// TIA Portal V17 program export: 1 tag tables, 0 data types, 4 data blocks, 2 code blocks (in call order from the OBs), 2 instance data blocks

VAR_GLOBAL   // PLC tag table "Tabla de variables estándar"
   System_Byte AT %MB1 : Byte;
   FirstScan AT %M1.0 : Bool;
   DiagStatusUpdate AT %M1.1 : Bool;
   AlwaysTRUE AT %M1.2 : Bool;
   AlwaysFALSE AT %M1.3 : Bool;
   Clock_Byte AT %MB0 : Byte;
   Clock_10Hz AT %M0.0 : Bool;
   Clock_5Hz AT %M0.1 : Bool;
   "Clock_2.5Hz" AT %M0.2 : Bool;
   Clock_2Hz AT %M0.3 : Bool;
   "Clock_1.25Hz" AT %M0.4 : Bool;
   Clock_1Hz AT %M0.5 : Bool;
   "Clock_0.625Hz" AT %M0.6 : Bool;
   "Clock_0.5Hz" AT %M0.7 : Bool;
   RISING_EDGE AT %M3.0 : Bool;
   INDEX AT %MB2 : USInt;
   MODE AT %MB6 : USInt;
   RISING_REQ AT %M3.1 : Bool;
   VOLTS AT %MW4 : UInt;
   AMPS AT %MW8 : UInt;
   HERTZ AT %MW10 : UInt;
   RPM AT %MW12 : UInt;
END_VAR
VAR_GLOBAL CONSTANT   // user constants
   READ : USInt := 0;
   WRITE : USInt := 1;
END_VAR

DATA_BLOCK "DB_MB_COMM_LOAD"   // DB4
{ S7_Optimized_Access := 'TRUE' }
VERSION : 0.1
// stored: AutoNumber true, DBAccessibleFromOPCUA true, IsOnlyStoredInLoadMemory false, IsRetainMemResEnabled false, IsWriteProtectedInAS false, MemoryReserve 100
   VAR
      COMM_DONE : Bool;
      COMM_ERROR : Bool;
      COMM_STATUS : Word;
   END_VAR
BEGIN
END_DATA_BLOCK

DATA_BLOCK "DB_ADDR"   // DB5
{ S7_Optimized_Access := 'FALSE' }
VERSION : 0.1
// stored: AutoNumber true, DBAccessibleFromOPCUA true, IsOnlyStoredInLoadMemory false, IsWriteProtectedInAS false
   VAR
      VOLT : UDInt := 48455;
      AMP : UDInt := 48453;
      FRE : UDInt := 48452;
      RPM : UDInt := 48456;
      SPEED : UDInt := 42331;
      RUN : UDInt := 42332;
      DIR : UDInt := 42333;
      OUT : UDInt;
   END_VAR
BEGIN
END_DATA_BLOCK

DATA_BLOCK "DB_GS1_MODBUS"   // DB6
{ S7_Optimized_Access := 'TRUE' }
VERSION : 0.1
// stored: AutoNumber true, DBAccessibleFromOPCUA true, IsOnlyStoredInLoadMemory false, IsRetainMemResEnabled false, IsWriteProtectedInAS false, MemoryReserve 100
   VAR
      GS1_DONE : Bool;
      GS1_BUSY : Bool;
      GS1_ERROR : Bool;
      GS1_STATUS : Word;
   END_VAR
BEGIN
END_DATA_BLOCK

DATA_BLOCK "DB_RW_PAR"   // DB3
{ S7_Optimized_Access := 'FALSE' }
VERSION : 0.1
// stored: AutoNumber true, DBAccessibleFromOPCUA true, IsOnlyStoredInLoadMemory false, IsWriteProtectedInAS false
   VAR
      VOLT_ACT : UInt;
      AMP_ACT : UInt;
      FRE_ACT : UInt;
      RPM_ACT : UInt;
      "SPEED(FREQ)" : UInt := 0;
      RUN : UInt := 0;
      DIR : UInt := 0;
      OUT : UInt;
   END_VAR
BEGIN
END_DATA_BLOCK

ORGANIZATION_BLOCK "Main"   // OB1, LAD, ProgramCycle
TITLE = "Main Program Sweep (Cycle)"
{ S7_Optimized_Access := 'TRUE' }
VERSION : 0.1
// stored: AutoNumber true, IsIECCheckEnabled false, SetENOAutomatically false
   VAR_INPUT
      Initial_Call : Bool;   // Initial call of this OB
      Remanence : Bool;   // =True, if remanent data are available
   END_VAR
BEGIN

REGION Network 1: ----------[MODBUS COMMUNICATION SETTING UP]----------
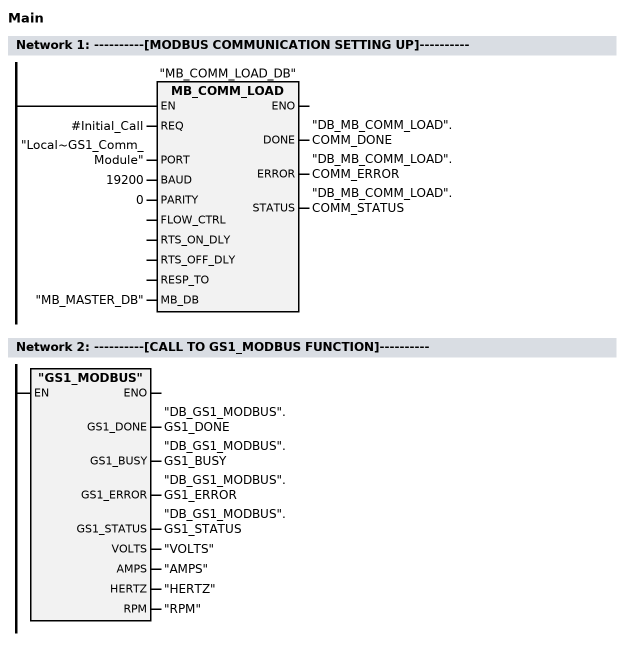
   RUNG wire#powerrail
      "MB_COMM_LOAD_DB".MB_COMM_LOAD(REQ := #Initial_Call, PORT := "Local~GS1_Comm_Module", BAUD := 19200, PARITY := 0, FLOW_CTRL :=, RTS_ON_DLY :=, RTS_OFF_DLY :=, RESP_TO :=, MB_DB := "MB_MASTER_DB", DONE => "DB_MB_COMM_LOAD".COMM_DONE, ERROR => "DB_MB_COMM_LOAD".COMM_ERROR, STATUS => "DB_MB_COMM_LOAD".COMM_STATUS)
   END_RUNG
   // the same network as SCL:
   "MB_COMM_LOAD_DB"(REQ := #Initial_Call,   // MB_COMM_LOAD
                     PORT := "Local~GS1_Comm_Module",
                     BAUD := 19200,
                     PARITY := 0,
                     MB_DB := "MB_MASTER_DB",
                     DONE => "DB_MB_COMM_LOAD".COMM_DONE,
                     ERROR => "DB_MB_COMM_LOAD".COMM_ERROR,
                     STATUS => "DB_MB_COMM_LOAD".COMM_STATUS);
END_REGION

REGION Network 2: ----------[CALL TO GS1_MODBUS FUNCTION]----------
   RUNG wire#powerrail
      "GS1_MODBUS"(GS1_DONE => "DB_GS1_MODBUS".GS1_DONE, GS1_BUSY => "DB_GS1_MODBUS".GS1_BUSY, GS1_ERROR => "DB_GS1_MODBUS".GS1_ERROR, GS1_STATUS => "DB_GS1_MODBUS".GS1_STATUS, VOLTS => "VOLTS", AMPS => "AMPS", HERTZ => "HERTZ", RPM => "RPM")
   END_RUNG
   // the same network as SCL:
   "GS1_MODBUS"(GS1_DONE => "DB_GS1_MODBUS".GS1_DONE,
                GS1_BUSY => "DB_GS1_MODBUS".GS1_BUSY,
                GS1_ERROR => "DB_GS1_MODBUS".GS1_ERROR,
                GS1_STATUS => "DB_GS1_MODBUS".GS1_STATUS,
                VOLTS => "VOLTS",
                AMPS => "AMPS",
                HERTZ => "HERTZ",
                RPM => "RPM");
END_REGION
END_ORGANIZATION_BLOCK

FUNCTION "GS1_MODBUS" : Void   // FC1, LAD
TITLE = FUNCTION FOR SEND THE MODE (R/W OF REGISTERS), MODBUS MODE, REGISTERS ADDRESS AND LOAD VALUES
{ S7_Optimized_Access := 'TRUE' }
VERSION : 0.1
// stored: AutoNumber true, IsIECCheckEnabled false, SetENOAutomatically false, UDAEnableTagReadback false
   VAR_OUTPUT
      GS1_DONE : Bool;
      GS1_BUSY : Bool;
      GS1_ERROR : Bool;
      GS1_STATUS : Word;
      VOLTS : UInt;
      AMPS : UInt;
      HERTZ : UInt;
      RPM : UInt;
   END_VAR
   VAR_TEMP
      RW : Int;
   END_VAR
   VAR_TEMP   // added for the SCL form of the ladder/FBD networks
      _w1 : Bool;
   END_VAR
BEGIN

REGION Network 1: ----------[GENERATE MODBUS ADDRESS & COMMAND DATA INDEX]----------
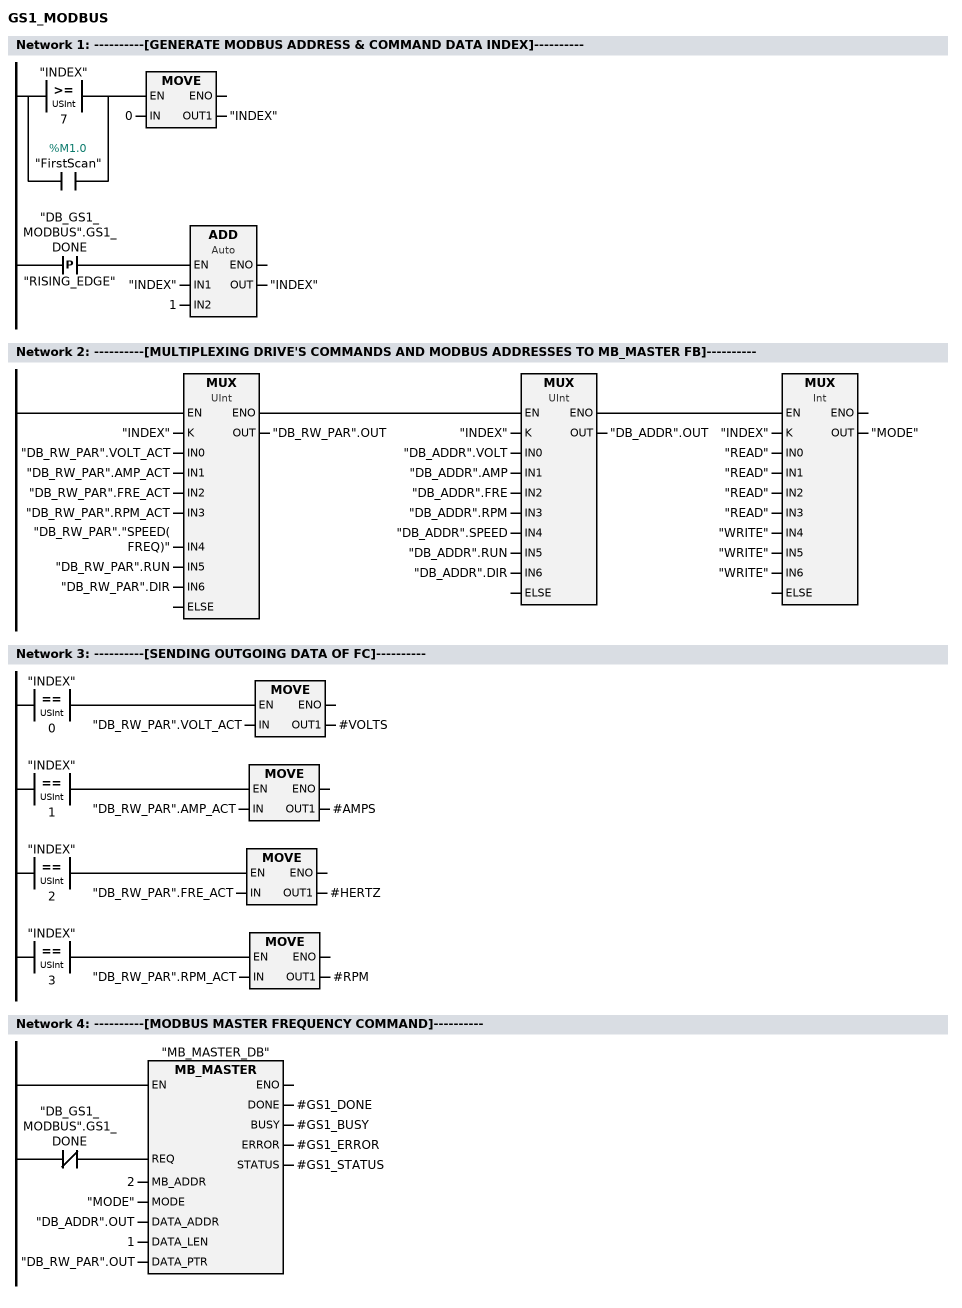
   RUNG wire#powerrail
      { S7_Templates := "SrcType := USInt" } GE_Contact(in1 := "INDEX", in2 := 7)
      wire#w1
      Move(in := 0, out1 => "INDEX")
   END_RUNG
   RUNG wire#powerrail
      Contact( "FirstScan" )
   END_RUNG wire#w1
   RUNG wire#powerrail
      P_Contact(operand := "DB_GS1_MODBUS".GS1_DONE, bit := "RISING_EDGE")
      Add(in1 := "INDEX", in2 := 1, out => "INDEX")
   END_RUNG
   // the same network as SCL:
   IF ("INDEX" >= 7) OR "FirstScan" THEN "INDEX" := 0; END_IF;
   #_w1 := "DB_GS1_MODBUS".GS1_DONE AND NOT "RISING_EDGE";   // rising edge of "DB_GS1_MODBUS".GS1_DONE
   "RISING_EDGE" := "DB_GS1_MODBUS".GS1_DONE;
   IF #_w1 THEN "INDEX" := "INDEX" + 1; END_IF;
END_REGION

REGION Network 2: ----------[MULTIPLEXING DRIVE'S COMMANDS AND MODBUS ADDRESSES TO MB_MASTER FB]----------
   RUNG wire#powerrail
      { S7_Templates := "SrcType := UInt"; S7_GenerateENO := "TRUE" } Mux(k := "INDEX", in0 := "DB_RW_PAR".VOLT_ACT, in1 := "DB_RW_PAR".AMP_ACT, in2 := "DB_RW_PAR".FRE_ACT, in3 := "DB_RW_PAR".RPM_ACT, in4 := "DB_RW_PAR"."SPEED(FREQ)", in5 := "DB_RW_PAR".RUN, in6 := "DB_RW_PAR".DIR, "else" :=, out => "DB_RW_PAR".OUT)
      { S7_Templates := "SrcType := UInt"; S7_GenerateENO := "TRUE" } Mux(k := "INDEX", in0 := "DB_ADDR".VOLT, in1 := "DB_ADDR".AMP, in2 := "DB_ADDR".FRE, in3 := "DB_ADDR".RPM, in4 := "DB_ADDR".SPEED, in5 := "DB_ADDR".RUN, in6 := "DB_ADDR".DIR, "else" :=, out => "DB_ADDR".OUT)
      { S7_Templates := "SrcType := Int"; S7_GenerateENO := "TRUE" } Mux(k := "INDEX", in0 := "READ", in1 := "READ", in2 := "READ", in3 := "READ", in4 := "WRITE", in5 := "WRITE", in6 := "WRITE", "else" :=, out => "MODE")
   END_RUNG
   // the same network as SCL:
   // no SCL statement known for Mux: written as a call
   // ENO of a box is taken as its EN; it also drops when the box reports an error
   Mux(k := "INDEX",
       in0 := "DB_RW_PAR".VOLT_ACT,
       in1 := "DB_RW_PAR".AMP_ACT,
       in2 := "DB_RW_PAR".FRE_ACT,
       in3 := "DB_RW_PAR".RPM_ACT,
       in4 := "DB_RW_PAR"."SPEED(FREQ)",
       in5 := "DB_RW_PAR".RUN,
       in6 := "DB_RW_PAR".DIR,
       out => "DB_RW_PAR".OUT);
   Mux(k := "INDEX",
       in0 := "DB_ADDR".VOLT,
       in1 := "DB_ADDR".AMP,
       in2 := "DB_ADDR".FRE,
       in3 := "DB_ADDR".RPM,
       in4 := "DB_ADDR".SPEED,
       in5 := "DB_ADDR".RUN,
       in6 := "DB_ADDR".DIR,
       out => "DB_ADDR".OUT);
   Mux(k := "INDEX",
       in0 := "READ",
       in1 := "READ",
       in2 := "READ",
       in3 := "READ",
       in4 := "WRITE",
       in5 := "WRITE",
       in6 := "WRITE",
       out => "MODE");
END_REGION

REGION Network 3: ----------[SENDING OUTGOING DATA OF FC]----------
   RUNG wire#powerrail
      { S7_Templates := "SrcType := USInt" } EQ_Contact(in1 := "INDEX", in2 := 0)
      Move(in := "DB_RW_PAR".VOLT_ACT, out1 => #VOLTS)
   END_RUNG
   RUNG wire#powerrail
      { S7_Templates := "SrcType := USInt" } EQ_Contact(in1 := "INDEX", in2 := 1)
      Move(in := "DB_RW_PAR".AMP_ACT, out1 => #AMPS)
   END_RUNG
   RUNG wire#powerrail
      { S7_Templates := "SrcType := USInt" } EQ_Contact(in1 := "INDEX", in2 := 2)
      Move(in := "DB_RW_PAR".FRE_ACT, out1 => #HERTZ)
   END_RUNG
   RUNG wire#powerrail
      { S7_Templates := "SrcType := USInt" } EQ_Contact(in1 := "INDEX", in2 := 3)
      Move(in := "DB_RW_PAR".RPM_ACT, out1 => #RPM)
   END_RUNG
   // the same network as SCL:
   IF "INDEX" = 0 THEN #VOLTS := "DB_RW_PAR".VOLT_ACT; END_IF;
   IF "INDEX" = 1 THEN #AMPS := "DB_RW_PAR".AMP_ACT; END_IF;
   IF "INDEX" = 2 THEN #HERTZ := "DB_RW_PAR".FRE_ACT; END_IF;
   IF "INDEX" = 3 THEN #RPM := "DB_RW_PAR".RPM_ACT; END_IF;
END_REGION

REGION Network 4: ----------[MODBUS MASTER FREQUENCY COMMAND]----------
   RUNG wire#powerrail
      "MB_MASTER_DB".MB_MASTER(REQ := wire#w1, MB_ADDR := 2, MODE := "MODE", DATA_ADDR := "DB_ADDR".OUT, DATA_LEN := 1, DATA_PTR := "DB_RW_PAR".OUT, DONE => #GS1_DONE, BUSY => #GS1_BUSY, ERROR => #GS1_ERROR, STATUS => #GS1_STATUS)
   END_RUNG
   RUNG wire#powerrail
      I_Contact( "DB_GS1_MODBUS".GS1_DONE )
   END_RUNG wire#w1
   // the same network as SCL:
   "MB_MASTER_DB"(REQ := NOT "DB_GS1_MODBUS".GS1_DONE,   // MB_MASTER
                  MB_ADDR := 2,
                  MODE := "MODE",
                  DATA_ADDR := "DB_ADDR".OUT,
                  DATA_LEN := 1,
                  DATA_PTR := "DB_RW_PAR".OUT,
                  DONE => #GS1_DONE,
                  BUSY => #GS1_BUSY,
                  ERROR => #GS1_ERROR,
                  STATUS => #GS1_STATUS);
END_REGION
END_FUNCTION

DATA_BLOCK "MB_COMM_LOAD_DB"   // DB1
// stored: AutoNumber true, DBAccessibleFromOPCUA true, InstanceOfName MB_COMM_LOAD, OfSystemLibElement MB_COMM_LOAD, OfSystemLibVersion 2.1
"MB_COMM_LOAD"
   // VAR_INPUT
   //    REQ : Bool;
   //    PORT : PORT;
   //    BAUD : UDInt;
   //    PARITY : UInt;
   //    FLOW_CTRL : UInt;
   //    RTS_ON_DLY : UInt;
   //    RTS_OFF_DLY : UInt;
   //    RESP_TO : UInt;
   // END_VAR
   // VAR_OUTPUT
   //    DONE : Bool;
   //    ERROR : Bool;
   //    STATUS : Word;
   // END_VAR
   // VAR_IN_OUT
   //    MB_DB : MB_BASE;
   // END_VAR
   // VAR
   //    ICHAR_GAP : UInt;
   //    RETRIES : UInt;
   //    WRREC_STATUS : Word;
   //    RDREC_STATUS : Word;
   //    SFC_STATUS : Word;
   //    Port_CFG_SFB : Array[0..25] of Byte;
   //    Send_CFG_SFB : Array[0..16] of Byte;
   //    Rcv_CFG_SFB : Array[0..60] of Byte;
   //    STOP_BITS : USInt;
   // END_VAR
BEGIN
END_DATA_BLOCK

DATA_BLOCK "MB_MASTER_DB"   // DB2
// stored: AutoNumber true, DBAccessibleFromOPCUA true, InstanceOfName MB_MASTER, OfSystemLibElement MB_MASTER, OfSystemLibVersion 2.2
"MB_MASTER"
   // // inherited from MB_BASE
   // VAR
   //    S_PORT : UInt;
   //    S_RESP_TO : UInt;
   //    S_ICHAR_GAP : UInt;
   //    S_RETRIES : UInt;
   // END_VAR
   // VAR_INPUT
   //    REQ : Bool;
   //    MB_ADDR : UInt;
   //    MODE : USInt;
   //    DATA_ADDR : UDInt;
   //    DATA_LEN : UInt;
   // END_VAR
   // VAR_OUTPUT
   //    DONE : Bool;
   //    BUSY : Bool;
   //    ERROR : Bool;
   //    STATUS : Word;
   // END_VAR
   // VAR_IN_OUT
   //    DATA_PTR : Variant;
   // END_VAR
   // VAR
   //    SEND_PTP_SFB : Array[0..11] of Byte;
   //    RCV_PTP_SFB : Array[0..11] of Byte;
   //    RCV_RST_SFB : Array[0..9] of Byte;
   //    PF_FREQUENCY : Real;
   //    BLOCKED_PROC_TIMEOUT : Real;
   //    CURRENT_TIME_VALUE : UDInt;
   //    SAVED_TIME_VALUE : UDInt;
   //    SAVED_SLAVE_ADDR : Word;
   //    SAVED_MODE : Word;
   //    SAVED_DATA_ADDR : DWord;
   //    SAVED_DATA_LEN : UInt;
   //    MB_STATE : UInt;
   //    COMM_SENT_COUNT : UInt;
   //    BYTE_COUNT : USInt;
   //    INIT_OK : Bool;
   //    ACTIVE : Bool;
   //    BROADCAST_FLAG : Bool;
   //    EXTENDED_ADDRESSING : Bool;
   //    SAVED_START_ADDR : UInt;
   //    TXBuf_Function_Offset : UDInt;
   //    TXBuf_Address_Offset : UDInt;
   //    TXBuf_Quantity_Offset : UDInt;
   // END_VAR
BEGIN
END_DATA_BLOCK
